PROGRAM BiogasProcess
VAR
	
(************** Pressure Sensor **************************************************)
	fbPressureSens_GH01	 : FB_Scaling; //Czujnik ciśnienia w  GH01
	

(************** Flow Sensor **************************************************)
	fbFlowSens_F01		 : FB_DigitalSensNO; //Czujnik poziomu cieczy w reaktorze R01

(************** Flow Counter **************************************************)	
   fbFlowCounter_F01	 : FB_FlowCounter;	


	fbMedian_PressureSens: FB_Median5;
END_VAR

ACT_PressureSens();
ACT_FlowSens();
ADS_BiogasTorch();

ACTION ACT_FlowSens:
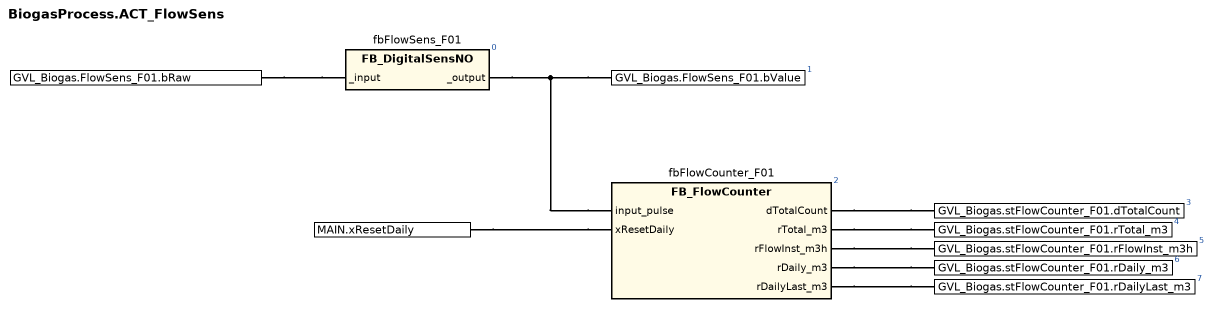
fbFlowSens_F01(_input := GVL_Biogas.FlowSens_F01.bRaw); // FB_DigitalSensNO
GVL_Biogas.FlowSens_F01.bValue := fbFlowSens_F01._output;
fbFlowCounter_F01(input_pulse := fbFlowSens_F01._output, xResetDaily := MAIN.xResetDaily); // FB_FlowCounter
GVL_Biogas.stFlowCounter_F01.dTotalCount := fbFlowCounter_F01.dTotalCount;
GVL_Biogas.stFlowCounter_F01.rTotal_m3 := fbFlowCounter_F01.rTotal_m3;
GVL_Biogas.stFlowCounter_F01.rFlowInst_m3h := fbFlowCounter_F01.rFlowInst_m3h;
GVL_Biogas.stFlowCounter_F01.rDaily_m3 := fbFlowCounter_F01.rDaily_m3;
GVL_Biogas.stFlowCounter_F01.rDailyLast_m3 := fbFlowCounter_F01.rDailyLast_m3;
END_ACTION

ACTION ACT_PressureSens:
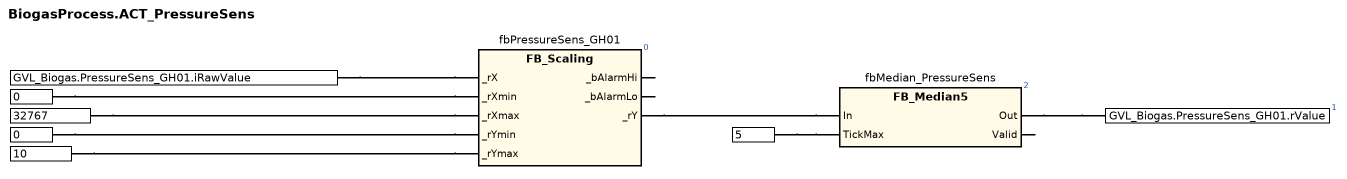
fbPressureSens_GH01(
    _rX := GVL_Biogas.PressureSens_GH01.iRawValue,
    _rXmin := 0,
    _rXmax := 32767,
    _rYmin := 0,
    _rYmax := 10); // FB_Scaling
GVL_Biogas.PressureSens_GH01.rValue := fbMedian_PressureSens.Out;
fbMedian_PressureSens(In := fbPressureSens_GH01._rY, TickMax := 5); // FB_Median5
END_ACTION

END_PROGRAM

(* stored: Version 1.1.0.1, ProductVersion 3.1.4024.16
   POU BiogasProcess: Id {42ee1a91-553f-4003-838c-56a71dec62fc}, SpecialFunc None
   Action ACT_FlowSens: Id {6fe933f2-7a93-4b42-ae83-e92ce890041a}
   Action ACT_PressureSens: Id {bb8a141f-b794-40f7-8523-14ae27fe1cf3} *)
